FUNCTION SPHERE_V : REAL
VAR_INPUT
	rx : REAL;
END_VAR


(*
version 1.2	22. feb 2008
programmer 	hugo
tested by		tobias

sphere_V calculates the Volume of a Sphere


*)

sphere_V := 4.188790205 * Rx * RX * RX;

(* revision histroy
hm	16. oct 2007	rev 1.0
	original version

hm	4. dec 2007		rev 1.1
	changed code for better performance

hm	22. feb 2008		rev 1.2
	changed code for better performance
*)

END_FUNCTION

(* stored: Version 1.1.0.1, ProductVersion 3.1.4024.9
   POU SPHERE_V: Id {fbdc0be5-64ca-4d50-8387-2dfb0b52bb8c}, SpecialFunc None *)
